TYPE "SSA_Germ_Par"	// UDT 2201
VERSION : 0.1
  STRUCT
   Switches1 : STRUCT
    StaOn24 : BOOL ;	//Example for comment: StaOn24WaterPumpA
    StaOn25 : BOOL ;
    StaOn26 : BOOL ;
    StaOn27 : BOOL ;
    StaOn28 : BOOL ;
    StaOn29 : BOOL ;
    StaOn30 : BOOL ;
    StaOn31 : BOOL ;
    StaOn16 : BOOL ;
    StaOn17 : BOOL ;
    StaOn18 : BOOL ;
    StaOn19 : BOOL ;
    StaOn20 : BOOL ;
    StaOn21 : BOOL ;
    StaOn22 : BOOL ;
    StaOn23 : BOOL ;
    StaOn08 : BOOL ;
    StaOn09 : BOOL ;
    StaOn10 : BOOL ;
    StaOn11 : BOOL ;
    StaOn12 : BOOL ;
    StaOn13 : BOOL ;
    StaOn14 : BOOL ;
    StaOn15 : BOOL ;
    StaOn00 : BOOL ;
    StaOn01 : BOOL ;
    StaOn02 : BOOL ;
    StaOn03 : BOOL ;
    StaOn04 : BOOL ;
    StaOn05 : BOOL ;
    StaOn06 : BOOL ;
    StaOn07 : BOOL ;
   END_STRUCT ;
   Switches2 : STRUCT
    StaOn24 : BOOL ;
    StaOn25 : BOOL ;
    StaOn26 : BOOL ;
    StaOn27 : BOOL ;
    StaOn28 : BOOL ;
    StaOn29 : BOOL ;
    StaOn30 : BOOL ;
    StaOn31 : BOOL ;
    StaOn16 : BOOL ;
    StaOn17 : BOOL ;
    StaOn18 : BOOL ;
    StaOn19 : BOOL ;
    StaOn20 : BOOL ;
    StaOn21 : BOOL ;
    StaOn22 : BOOL ;
    StaOn23 : BOOL ;
    StaOn08 : BOOL ;
    StaOn09 : BOOL ;
    StaOn10 : BOOL ;
    StaOn11 : BOOL ;
    StaOn12 : BOOL ;
    StaOn13 : BOOL ;
    StaOn14 : BOOL ;
    StaOn15 : BOOL ;
    StaOn00 : BOOL ;
    StaOn01 : BOOL ;
    StaOn02 : BOOL ;
    StaOn03 : BOOL ;
    StaOn04 : BOOL ;
    StaOn05 : BOOL ;
    StaOn06 : BOOL ;
    StaOn07 : BOOL ;
   END_STRUCT ;
   Values1 : STRUCT 	//Lineparameter data written by Host-System
    Value01 : DINT ;	//Example for comment: TurnoverTime [xxxs]
    Value02 : DINT ;
    Value03 : DINT ;
    Value04 : DINT ;
    Value05 : DINT ;
    Value06 : DINT ;
    Value07 : DINT ;
    Value08 : DINT ;
    Value09 : DINT ;
    Value10 : DINT ;
    Value11 : DINT ;
    Value12 : DINT ;
    Value13 : DINT ;
    Value14 : DINT ;
    Value15 : DINT ;
    Value16 : DINT ;
    Value17 : DINT ;
    Value18 : DINT ;
    Value19 : DINT ;
    Value20 : DINT ;
    Value21 : DINT ;
    Value22 : DINT ;
    Value23 : DINT ;
    Value24 : DINT ;
    Value25 : DINT ;
    Value26 : DINT ;
    Value27 : DINT ;
    Value28 : DINT ;
    Value29 : DINT ;
    Value30 : DINT ;
   END_STRUCT ;
   FlagSec : STRUCT
    Flag00 : BOOL ;
    Flag001 : BOOL ;
    Flag002 : BOOL ;
    Flag003 : BOOL ;
    Flag004 : BOOL ;
    Flag005 : BOOL ;
    Flag006 : BOOL ;
    Flag007 : BOOL ;
    Flag008 : BOOL ;
    Flag009 : BOOL ;
    Flag0010 : BOOL ;
    Flag0011 : BOOL ;
    Flag0012 : BOOL ;
    Flag0013 : BOOL ;
    Flag0014 : BOOL ;
    Flag0015 : BOOL ;
    Flag0016 : BOOL ;
    Flag0017 : BOOL ;
    Flag0018 : BOOL ;
    Flag0019 : BOOL ;
    Flag0020 : BOOL ;
    Flag0021 : BOOL ;
    Flag0022 : BOOL ;
    Flag0023 : BOOL ;
    Flag0024 : BOOL ;
    Flag0025 : BOOL ;
    Flag0026 : BOOL ;
    Flag0027 : BOOL ;
    Flag0028 : BOOL ;
    Flag0029 : BOOL ;
    Flag0030 : BOOL ;
    Flag0031 : BOOL ;
   END_STRUCT ;
   FlagGen : STRUCT
    WindAlarm : BOOL ;	//Wind speed is too high
    TurningStarted : BOOL ;	//Germination turning is started
    Underhorden_Clean_aktiv : BOOL ;	//Unterhordenreinigung aktiv
    WetStep : BOOL ;	//Active Step is Wet Step
    Flag004 : BOOL ;
    Flag005 : BOOL ;
    Flag006 : BOOL ;
    Flag007 : BOOL ;
    LOAD_VAL_HUB1 : BOOL ;	//Counter lifting device 1
    LOAD_VAL_HUB2 : BOOL ;	//Counter lifting device 2
    LOAD_VAL_DRIVE : BOOL ;	//Counter driving device
    LOAD_VAL_AFTER_FAILURE : BOOL ;	//Counter saved datas after failure
    Flag0012 : BOOL ;
    Flag0013 : BOOL ;
    Flag0014 : BOOL ;
    Flag0015 : BOOL ;
    InterlockedFunktionMode : BOOL ;
    ILO_CmdResetFault : BOOL ;
    Flag0018 : BOOL ;
    Flag0019 : BOOL ;
    Flag0020 : BOOL ;
    Flag0021 : BOOL ;
    Flag0022 : BOOL ;
    Flag0023 : BOOL ;
    Flag0024 : BOOL ;
    Flag0025 : BOOL ;
    Flag0026 : BOOL ;
    Flag0027 : BOOL ;
    Flag0028 : BOOL ;
    Flag0029 : BOOL ;
    Flag0030 : BOOL ;
    Flag0031 : BOOL ;
   END_STRUCT ;
   Spare140 : ARRAY  [148 .. 194 ] OF BYTE ;
   FlagMachine_0 : STRUCT 	//flags machine funktion
    FloorFwdPlus : BOOL ;	//Hordendrehrichtung Vorwärts, Rundenzaehler +1
    FloorFwdMinus : BOOL ;	//Hordendrehrichtung Vorwärts, Rundenzaehler -1
    FloorRevPlus : BOOL ;	//Hordendrehrichtung Rückwärts, Rundenzaehler +1
    FloorRevMinus : BOOL ;	//Hordendrehrichtung Rückwärts, Rundenzaehler -1
    OneShotGeenVrygVlr : BOOL ;	//Opkomende Flank geen vrijgave vloer
    HulpOneShotGeenVrygVlr : BOOL ;	//Hulp Opkomende Flank geen vrijgave vloer
    Flag006 : BOOL ;	//
    Flag007 : BOOL ;	//
    RotatPulseNotZero : BOOL ;	//
    ReducedSpeed : BOOL ;	//
    Speed2ndRound : BOOL ;	//Speed 2nd round during loading
    Flag013 : BOOL ;	//
    Flag014 : BOOL ;	//
    Flag015 : BOOL ;	//
    Flag016 : BOOL ;	//
    Flag017 : BOOL ;	//
    Flag020 : BOOL ;	//
    Flag021 : BOOL ;	//
    Flag022 : BOOL ;	//
    Flag023 : BOOL ;	//
    Flag024 : BOOL ;	//
    Flag025 : BOOL ;	//
    Flag026 : BOOL ;	//
    Flag027 : BOOL ;	//
    Flag030 : BOOL ;	//
    Flag031 : BOOL ;	//
    Flag032 : BOOL ;	//
    Flag033 : BOOL ;
    Flag034 : BOOL ;
    Flag035 : BOOL ;
    Flag036 : BOOL ;	//
    Flag037 : BOOL ;	//
   END_STRUCT ;
   ParIntProcess : STRUCT 	//Processparameter data
    UnloadungRounds : INT  := 2;
    LoadungRounds : INT  := 2;	//
    LoadingOverlap : INT  := 10;	//Impulse overlap by loading
    UnloadingOverlap : INT  := 20;	//Impulse overlap by unloading
    ReactTimeTempContr : S5TIME  := S5T#10S;	//Delay reaction temperature control below floor
    ReactTimeCO2Contr1 : S5TIME  := S5T#10S;	//Delay reaction CO2 control below floor
    BreakTimeFlapContr1 : S5TIME  := S5T#10S;	//Break time control fresh air flap
    DelayContrDelta_T : INT  := 10;	//Delay alarm control Delta-t in min
    DelayDeltaTemp : INT  := 2;	//Delay control Delta-t between temperature above and below floor, in min
    DelayMaxTemp : INT  := 2;	//Delay control temperature above below floor, in min
    Speed_ILO_FloorRotating : INT  := 22;	//Rotating speed floor from ILO-Rotating Floor Drives
    Speed_ILO_UnderCleaning : INT  := 80;	//Rotating speed floor from ILO-Floor Cleaning from below
    Speed_ILO_WallCleaning : INT  := 80;	//Rotating speed floor from ILO-WallCleaning
    ProcessActivVisuGerm : INT ;	//Display that Process is Active
    StateWordGerm : INT ;	//State-Number of the active Step
    TarPos_ILO_LiftDev : INT ;	//Target positon lifting devices from ILO-Mode
    TarPos_ILO_FreshAir : INT ;	//Target positon fresh air flap from ILO-Mode
    TarPos_ILO_RecycAir : INT ;	//Target positon recycling air flap from ILO-Mode
    Speed_ILO_Fan : INT ;	//Target speed germinatimng fan from ILO-Mode
    Speed_ILO_TravelDrive : INT ;	//Target speed travelling drive from ILO-Mode
    TarPos_ILO_WasteAir : INT ;	//Target positon waste air flap from ILO-Mode
    TargetTemperature_ILO : INT ;	//Target temperature from ILO-Mode
    Value23 : INT ;
    Value24 : INT ;
    Value25 : INT ;
    Value26 : INT ;
    Value27 : INT ;
    Value28 : INT ;
    Value29 : INT ;
    Value30 : INT ;
    Value31 : INT ;
    NextLevelLoading : INT ;	//Next level loading round
    Value33 : INT ;
    Value34 : INT ;
    Value35 : INT ;
    Value36 : INT ;
    CounterPosLoadingBeam : INT ;	//external counter beam position
    Value38 : INT ;
    Value39 : INT ;
    NumberOpenValves : INT ;	//number of opened spray valves air humidifikation
    SpeedProdSprayPump : INT ;	//setpoint speed pump product spray
    Value42 : INT ;
    Value43 : INT ;
    Value44 : INT ;
    PrevStep1stTurn : INT ;	//Store turning commands from prev. step
    PrevStep2ndTurn : INT ;	//Store turning commands from prev. step
    Value47 : INT ;
    Value48 : INT ;
    Value49 : INT ;
    ActualStep : INT ;	//Actual Step for visu
   END_STRUCT ;
   ParIntMachine : STRUCT 	//Machine parameter data
    ActualStep : INT ;	//Actual process step
    MAX_HUB_DIFF : INT  := 36;	//Max. Hubdifferenz zwischen Hubzug 1 + 2
    REINIGUNGSHOEHE : INT  := 100;	//Reinigungshoehe in mm
    MAX_SCHIEFLAGE : INT  := 150;	//Max. Schieflage zwischen Hubzug 1 + 2
    IMPULSE_HUBZUG1_OBEN : INT  := 480;	//Impulse : Hubantrieb 1 normieren bei Endpos.oben
    IMPULSE_HUBZUG2_OBEN : INT  := 480;	//Impulse : Hubantrieb 2 normieren bei Endpos.oben
    POSITION_HUBZUG1_OBEN : INT  := 1055;	//Hoehe in mm
    POSITION_HUBZUG2_OBEN : INT  := 1055;	//Hoehe in mm
    IMPULSE_RUNDE : INT  := 816;	//Impulse : Fahrantriebantrieb eine Runde (Diesen Wert bei der IBS ermitteln!!)
    SollwertFahrantrWenden : WORD  := W#16#DEF;	//21,7% von 100 Hz
    LiftDevMinPos : INT  := 100;	//Lifting device minimal position for rotation backwards
    FUELLHOEHE_PRODUKT : INT ;	//Produkt-Füllhöhe
    TargetPosTravDriveLoad : INT ;	//Soll-Position Fahrantrieb im Prozess
    RunTimeCleanDrive : S5TIME  := S5T#10M;	//Runing time drive floor cleaning from below
    DelayMonFlowContr : S5TIME  := S5T#10M;	//Delay monitoring flow control by loading
    RunTimeTurnScrews : INT  := 2;	//Time short run turning screws every 6 hours, in min
    LiftDevLowPos : INT  := 1000;	//Lifting device lowered position after turning round, in mm
    CutOffPointDosing : INT ;	//Cut-off point dosing
    GerminatingBoxNumber : INT ;
    TargetPosTravDriTurnLeft : INT ;
    TargetPosTravDriTurnRigt : INT ;
    TargetPosTravDriveUnload : INT ;
    Help1StartTurning : INT ;	//hulpwoord 1 tbv  wenderen
    Resetbreaktime : INT ;	//tbv resetten wenderpauze
    Help2StartTurning : INT ;	//hulpwoord 2 tbv  wenderen
    TurningHourOneOrTwo : INT ;	//wenderuur 1 of 2
    Timer_tbv_opk_wend_spr : INT ;	//timer tbv het opkomen van het wenderen of sproeien
    TargetPosFreshAir : INT ;	//Target position fresh air flap/jalousie/louver
    TargetPosRecyclingAir : INT ;	//Target position recycling air flap/jalousie/louver
    TargetPosWasteAir : INT ;	//Target position waste air flap/jalousie/louver
    TargetSpeedGermFan : INT ;	//Target speed fan germinating box
    TargetSpeedLoadScrew : INT ;	//Target speed loading/unloading screw germinating box
    Value33 : INT ;
    Value34 : INT ;
    Value35 : INT ;
    Value36 : INT ;
    Value37 : INT ;
    HulpwoordTbvTelpulsbewak : INT ;	//Hulpwoord tbv telpulsbewaking vloer
    PresetWaardeTimerTelpVlR : INT ;	//Preset waarde van timer tbv telpulsbewaking vloer.
    GemiddeldeHoogteHefwerk : INT ;	//De gemiddelde hoogte van de hefwerken
    GewensteOntlaadhoogte : INT ;	//Gewenste Ontlaadhoogte Hefwerken
    Value42 : INT ;
    Value43 : INT ;
    Value44 : INT ;
    Value45 : INT ;
    Value46 : INT ;
    Value47 : INT ;
    Value48 : INT ;
    GrowingOffset : INT ;
    LastLoadingLevel : INT ;
   END_STRUCT ;
   FlagFunction_0 : STRUCT 	//Flags section
    FlagLoadingFinishedFP : BOOL ;	//
    FlagFirstTurning : BOOL ;	//First turning round after loading
    FlagNextStep : BOOL ;
    FlagLoadingFinished : BOOL ;
    StartTurningForMGR : BOOL ;	//Enable start turning for group control
    Inf29 : BOOL ;
    FlagLoadingOverlap : BOOL ;
    FlagUnloadingOverlap : BOOL ;
    ImpulsUnloadLevelReached : BOOL ;	//Unloading level has been reached
    UnloadLevelReachedFP : BOOL ;	//FP unloading level has been reached
    ShortRunTurnScrews : BOOL ;	//Short run turning screws every 6 hours
    LowerLiftDevAfterTurn : BOOL ;	//To lower lifting device after every turning round
    UnloadingLevelAdjusted : BOOL ;	//
    FlagWallCleanStopFP : BOOL ;	//
    Spare2 : BOOL ;	//
    FlagLoadingStartedFP : BOOL ;
    ImpulseLoadingStarted : BOOL ;
    FlagUnloadingStartedFP : BOOL ;
    ImpulseUnloadingStarted : BOOL ;
    FlagCleaningStartedFP : BOOL ;
    ImpulseCleaningStarted : BOOL ;
    FlagTurningStartedFP : BOOL ;
    ImpulseTurningStarted : BOOL ;
    FlagTurningStartedRight : BOOL ;
    FlagTurningStartedLeft : BOOL ;
    FlagStep14FN : BOOL ;
    ImpulseUnloadFirstPart : BOOL ;
    FlagStepFirstTurning : BOOL ;	//First turning round in this step is finished
    FlagStepSecondTurning : BOOL ;	//Second turning round in this step is finished
    ReleaseUnloadFirstPart : BOOL ;
    InfReleaseUnloading : BOOL ;
   END_STRUCT ;
   FlagMachine : STRUCT 	//flags machine funktion
    Hubzug1_Low : BOOL ;	//Hubzug 1 Richtungsvorwahl senken
    Hubzug1_High : BOOL ;	//Hubzug 1 Richtungsvorwahl heben
    Hubzug2_Low : BOOL ;	//Hubzug 2 Richtungsvorwahl senken
    Hubzug2_High : BOOL ;	//Hubzug 2 Richtungsvorwahl heben
    Stop_Hubzuege : BOOL ;	//Differenz Hub1-Hub2>Vorgabewert
    Hubzug1_Speed_Ctr : BOOL ;	//Hubantrieb 1 innen Drehueberwachung
    Hubzug2_Speed_Ctr : BOOL ;	//Hubantrieb 2 aussen Drehueberwachung
    Hubzuege_ueber_MinPos : BOOL ;	//Hubzug 1 und Hubzug 2 mehr als 100mm ueber ihrer Nullposition
    Hubzug1_Stop_NullPos_man : BOOL ;	//Hoehe Hubzug 1 <= NULL-Position
    Hubzug2_Stop_NullPos_man : BOOL ;	//Hoehe Hubzug 2 <= NULL-Position
    Hubdiff1_2 : BOOL ;	//Hubdifferenz Hub1 > Hub2
    Hubdiff2_1 : BOOL ;	//Hubdifferenz Hub2 > Hub1
    Hubzug1_Hoch : BOOL ;	//Hubzug 1 Isthoehe > 300mm (Freigabe Ausraeumglocke schliessen) und Hubzuege heb
    Hubzug2_Hoch : BOOL ;	//Hubzug 2 Isthoehe > 300mm (Freigabe Ausraeumglocke schliessen) und Hubzuege heb
    Start_Hubzuege_Heben : BOOL ;	//Hubzuege heben
    Hubdiff1_2_NegAlt : BOOL ;	//Hubdifferenz Hub1 > Hub2 Alt-Signal
    Hubdiff1_2_NegFlag : BOOL ;	//Hubdifferenz Hub1 > Hub2 Flanken-Signal
    Hubdiff2_1_NegAlt : BOOL ;	//Hubdifferenz Hub2 > Hub1 Alt-Signal
    Hubdiff2_1_NegFlag : BOOL ;	//Hubdifferenz Hub2 > Hub1 Flanken-Signal
    Fahrantrieb_Speed_Ctr1 : BOOL ;	//Fahrantrieb Drehueberwachung
    Fahrantrieb_Start_ok : BOOL ;	//Es sind weniger als 2 Fahrantriebe nicht gestartet
    Fahrantrieb_FU_Fault : BOOL ;	//Sammelstörung von allen 12 FU's
    Fahrantriebe_Fwd_Rev : BOOL ;	//Aktuelle Drehrichtung Fahrantriebe (0=Fwd; 1=Rev)
    Fahrantriebe_Vorwaerts : BOOL ;	//Fahrantriebe Ausgang Richtung Vorwärts
    Fahrantriebe_Rueckwaerts : BOOL ;	//Fahrantriebe Ausgang Richtung Rückwärts
    NULL_INDEX_FP : BOOL ;
    ImpulsNullstellung : BOOL ;
    ImpulsNullstellungFP : BOOL ;
    WEGMESSUNG_0 : BOOL ;
    WEGMESSUNG_0_FLAG : BOOL ;
    HubzuegeUeberProdukt : BOOL ;	//Schnecke ueber Produktschicht
    HubzuegeParkposition : BOOL ;	//Beide Hubzuege in Parkposition
   END_STRUCT ;
   FlagFunction_1 : STRUCT 	//Flags functions
    StepLoading : BOOL ;	//Function Loading is active
    StepUnloading : BOOL ;	//Function Unloading is active
    StepCleaning : BOOL ;	//Function Cleaning is active
    LoadingBreak : BOOL ;	//Function Loading is interrupted
    UnloadingBreak : BOOL ;	//Function Unloading is interrupted
    CleaningBreak : BOOL ;	//Function Cleaning is interrupted
    FinishLoading : BOOL ;	//Function Loading is finished
    FinishUnloading : BOOL ;	//Function Unloading is finished
    FinishCleaning : BOOL ;	//Function Cleaning is finished
    LoadingStarted : BOOL ;	//Germination loading is started
    UnloadingStarted : BOOL ;	//Germination unloading is started
    CleaningStarted : BOOL ;	//Germination cleaning is started
    Round_1 : BOOL ;	//Fahrantrieb 1.Runde
    Round_2 : BOOL ;	//Fahrantrieb 2.Runde
    Round_3 : BOOL ;	//Fahrantrieb 3.Runde
    Round_4 : BOOL ;	//Fahrantrieb 4.Runde
    Round_5 : BOOL ;	//Fahrantrieb 5.Runde
    Round_6 : BOOL ;	//Fahrantrieb 6.Runde
    Beladung_beendet : BOOL ;	//Fahrantrieb; Beladung_beendet
    Entladerunden_erreicht : BOOL ;	//Fahrantrieb; Entladerunden erreicht
    Reinigungsrunde_erreicht : BOOL ;	//Fahrantrieb; Reinigungsrunde erreicht
    TurningStart : BOOL ;	//Start turning
    TurningStop : BOOL ;	//Stop turning
    TurningLeft : BOOL ;	//Germination turning left
    TurningRight : BOOL ;	//Germination turning right
    LoadFirstPartEnd : BOOL ;	//Grundschicht ist bedeckt, prozess kann starten
    TurningWithSpraying : BOOL ;	//Turning-round in this step with spraying
    TurningWithoutSpraying : BOOL ;	//Turning-round in this step without spraying
    UnloadFirstPartEnd : BOOL ;	//First half of germinating box is unloaded
    UnloadSecondPartEnd : BOOL ;	//Second half of germinating box is unloaded
    UnloadFirstPart : BOOL ;	//Unload first half of germinating box
    UnloadSecondPart : BOOL ;	//Unload second half of germinating box
   END_STRUCT ;
   FlagProcess : STRUCT 	//Flags process
    ProcessActive : BOOL ;	//Process is active
    ProcessStartFP : BOOL ;	//Flank start process
    ProcessStartScan : BOOL ;	//Impulse first step
    MessageNoNextStep : BOOL ;	//Message "No next step"
    FP_SendResultToPIC : BOOL ;
    Vraag_menu_wenderen : BOOL ;	//Vraag vanuit het recept om te wenderen
    Vraag_menu_sproeien : BOOL ;	//Vraag vanuit het recept om te sproeien
    Vraag_menu_doseren : BOOL ;	//Vraag vanuit het recept om te doseren
    FlagWallCleanStartFP : BOOL ;	//Hulp one shot wandreinigen gestart
    ImpulseWallCleanStarted : BOOL ;	//One shot wandreinigen gestart
    Inf18 : BOOL ;
    VrijgaveWenderFunctie : BOOL ;	//Geen vrijgave om wenderbits in FC2019 aan te zetten
    Aussenluft_zu_warm : BOOL ;
    Cooling : BOOL ;
    AirHumidificationValve1 : BOOL ;
    AirHumidificationValve2 : BOOL ;
    Breakpoint_Aktiv : BOOL ;
    ProcessEnd : BOOL ;
    Cooling_Activ : BOOL ;
    Abkuehlen : BOOL ;
    Inf24 : BOOL ;
    Vent_ReglerAusg_Plus : BOOL ;
    Vent_ReglerAusg_PlusFP : BOOL ;
    Vent_ReglerAusg_Minus : BOOL ;
    Vent_ReglerAusg_MinusFP : BOOL ;
    Ventilator_Drehzahl_HH : BOOL ;	// Drehzahlbereich HH [85 - 100%]
    Ventilator_Drehzahl_H : BOOL ;	// Drehzahlbereich  H [65 -  84%]
    Ventilator_Drehzahl_L : BOOL ;	// Drehzahlbereich  L [55 -  64%]
    Ventilator_Drehzahl_LL : BOOL ;	// Drehzahlbereich LL [40 -  54%]
    VentilatorDrehzahlMin : BOOL ;
    VentilatorDrehzahlMax : BOOL ;
    Inf37 : BOOL ;
   END_STRUCT ;
   FlagProcess1 : STRUCT 	//Flags process
    FreshAirFlapCLOSE : BOOL ;	//Close fresh air flap
    FreshAirFlapOPEN : BOOL ;	//Open fresh air flap
    ControlFreshAirFlap : BOOL ;	//Control fresh air flap
    ControlFlap_OPEN : BOOL ;	//Control - fresh air flap 1% open
    ControlFlap_CLOSE : BOOL ;	//Control - fresh air flap 1% close
    ControlTemperature : BOOL ;	//Priority temperature for control fresh air flap
    ControlCO2 : BOOL ;	//Priority CO2 for control fresh air flap
    BasicPosFreshAirFlap : BOOL ;	//Fresh air flap in basic position
    ExhaustAirFlap_1_CLOSE : BOOL ;	//Close exhaust air flap 1
    ExhaustAirFlap_1_OPEN : BOOL ;	//Open exhaust air flap 1
    BasicPosExhaustAirFlap_1 : BOOL ;	//Exhaust air flap 1 in basic position
    ExhaustAirFlap_2_CLOSE : BOOL ;	//Close exhaust air flap 2
    ExhaustAirFlap_2_OPEN : BOOL ;	//Open exhaust air flap 2
    BasicPosExhaustAirFlap_2 : BOOL ;	//Exhaust air flap 2 in basic position
    DeltaTempPlus : BOOL ;	//
    DeltaTempMinus : BOOL ;	//
    InterlockedFunktionMode : BOOL ;	//
    Inf21 : BOOL ;	//
    Inf22 : BOOL ;	//
    Inf23 : BOOL ;	//
    Inf24 : BOOL ;	//
    Inf25 : BOOL ;	//
    DeltaTempNextStep : BOOL ;	//Delta Temperature go to next step
    MaxTempNextStep : BOOL ;	//Max Temperature above floor go to next step
    FlankeStartRecept_IN : BOOL ;	//ONE_SHOT_START_RECEPT
    PT100Defect_IN : BOOL ;	//PT100_boven_vloer_stuk
    FreigabeStartRezept_IN : BOOL ;	//VRIJGAVE_START_RECEPT
    tm_Frequenzregler_IN : BOOL ;	//wanneer ventilator in bedrijf meldt
    Flanke_FreigabeRezept_IO : BOOL ;	//One_shot_vent_op_basis
    HandAutoVentilator_IO : BOOL ;	//Hand_automaat_kiemvent
    Inf36 : BOOL ;	//
    TurnWithClean : BOOL ;	//Turning with floor cleaning from below
   END_STRUCT ;
   FlagProcess2 : STRUCT 	//Flags process
    Turning1WithSpraying : BOOL ;	//First turning round in this step with spraying
    Turning1WithDosing : BOOL ;	//First turning round in this step with spraying and dosing
    Turning1WithoutSpraying : BOOL ;	//First turning round in this step without spraying
    Turning2WithSpraying : BOOL ;	//Second turning round in this step with spraying
    Turning2WithDosing : BOOL ;	//Second turning round in this step with spraying and dosing
    Turning2WithoutSpraying : BOOL ;	//Second turning round in this step without spraying
    MinBreakTimeFinish : BOOL ;	//Minimal break time is finished
    MaxBreakTimeFinish : BOOL ;	//Maximal break time is finished
    ReleaseSpraying : BOOL ;	//Release spraying for this germinating box
    ReleaseDosing : BOOL ;	//Release dosing for this germinating box
    Delta_T : BOOL ;	//Delta-t is > or < recipe value
    StartSpraying : BOOL ;	//Store impulse start spraying
    HighWindForce : BOOL ;	//Wind force too high
    ReleaseTurning : BOOL ;	//Release turning for this germinating box
    StartFirstTurningRound : BOOL ;	//Store impulse for start first turning round acc. recipe
    StartSecondTurningRound : BOOL ;	//Store impulse for start second turning round acc. recipe
    PauseBeforeSpraying_FP : BOOL ;	//
    PauseBeforeSpraying_IMP : BOOL ;
    PauseBeforeSprayingFin : BOOL ;	//Pause before spraying is finished
    AlarmControlDelta_T : BOOL ;	//Alarm control Delta-t
    StartFirstTurningFP : BOOL ;
    StartSecondTurningFP : BOOL ;	//
    StartFirstSprayingFP : BOOL ;
    StartFirstDosingFP : BOOL ;
    StartSecondSprayingFP : BOOL ;
    StartSecondDosingFP : BOOL ;
    StartFirstSpraying : BOOL ;	//Store impulse for start first turning round with spraying acc. recipe
    StartFirstDosing : BOOL ;	//Store impulse for start first turning round with dosing acc. recipe
    StartSecondSpraying : BOOL ;	//Store impulse for start second turning round with spraying acc. recipe
    StartSecondDosing : BOOL ;	//Store impulse for start second turning round with dosing acc. recipe
    Sonderwenden : BOOL ;	//Sonderwenden
    FaultDB_Copy : BOOL ;	//Fault DB Copy FC49
   END_STRUCT ;
   ProcessValue : STRUCT 	//Process values, used only in the PLC
    Value01 : DINT ;
    Value02 : DINT ;
    Value03 : DINT ;
    SetpointDeltaTempDint : DINT ;
    ActValueDeltaTempDint : DINT ;
    ActValMaxTempAboveDint : DINT ;
    ResultDeltaTemp : DINT ;
    ConsumptionWater : DINT ;	//Water consumption per section
    CurrentConsumCoolEnergy : DINT ;	//Aktueller Verbrauch Kühl-Energie
    ConsumptionCoolingEnergy : DINT ;	//Verbrauchte Menge Kühl-Energie
    LevelGlycol : DINT ;	//something with glycol
    Profimess_Command : DINT ;	//command to read data from Profimess
    Value13 : DINT ;
    Value14 : DINT ;
    Value15 : DINT ;
    Value16 : DINT ;
    HelpConsumptionwater : DINT ;	//Tussenwoord voor opslag aantal M3 sproeien
    RET_VAL_BreakTime : INT ;
    StepNrActCopy : INT ;
    StartStepAct : DATE_AND_TIME ;
    ActualTime : DATE_AND_TIME ;
    BreakTime : DATE_AND_TIME ;
    StartCooling : DATE_AND_TIME ;
    StepTimeAct : TIME ;
    BreakTimeAct : TIME ;
    TimeControlDelta_T : TIME ;
    PauseBeforeSpraying : TIME ;
   END_STRUCT ;
   ProcessValueReal : STRUCT 	//Process real values, used only in the PLC
    SpeedVentilatorBasic : REAL ;	//Setpoint Fanspeed in %
    PositFreshAirFlapBasic : REAL ;	//Setpoint basic flap position
    ActTempBelowFloor : REAL ;	//Actual temperature below floor
    TargTempBelowFloor : REAL ;	//Setpoint temperature below floor
    ActTempAboveFloor : REAL ;	//Actual temperature above floor
    TargTempAboveFloor : REAL ;	//Setpoint temperature above floor
    NivoDoseertank : REAL ;	//Nivo doseertank in real
    Value08 : REAL ;	//
    Value09 : REAL ;	//
    Value10 : REAL ;	//
    Value11 : REAL ;	//
    Value12 : REAL ;	//
    Value13 : REAL ;	//
    Value14 : REAL ;
    Value15 : REAL ;
    Value16 : REAL ;
    Value17 : REAL ;
    Value18 : REAL ;
    Value19 : REAL ;
    Value20 : REAL ;
    CoolingEnergyAct : REAL ;
    CoolingEnergySum : REAL ;
    Value23 : REAL ;
    Value24 : REAL ;
    Profimess_Wirkleistung : REAL ;
    Profimess_Blindleistung : REAL ;
    Profimess_Frequenz : REAL ;
    Profimess_Wirkleist_Psec : REAL ;
    Profimess_Arbeit_Batch : REAL ;
    EnergieKWs : REAL ;
   END_STRUCT ;
   MachineValue : STRUCT 	//Machine values, used only in the PLC
    ISTWERT_FAHRANTRIEB_POSI : INT ;	//Ist-Position Fahrantrieb
    FAHRANTRIEB_UMDREHUNGEN : INT ;	//Rundenzaehler Fahrantrieb
    IST_HUB_DIFF : INT ;	//Istwert Hubdifferenz zwischen Hubzug 1 + 2
    ISTWERT_HUBZUG1_Z_IMP : INT ;	//Istwert Zaehlimpulse Hubzug 1
    ISTWERT_HUBZUG2_Z_IMP : INT ;	//Istwert Zaehlimpulse Hubzug 2
    SCHRAEGE_HUB1_HUB2 : INT ;	//Schraege Hub 1 > Hub 2
    SOLLWERT_HUBZUG1_HOEHE : INT ;
    SOLLWERT_HUBZUG2_HOEHE : INT ;
    ISTWERT_HUBZUG1_HOEHE : INT ;
    ISTWERT_HUBZUG2_HOEHE : INT ;
    SCHRAEGE_HUB1_MINUS_HUB2 : INT ;	//Schraege Hub 1 minus Hub 2
    SCHRAEGE_HUB2_MINUS_HUB1 : INT ;	//Schraege Hub 2 minus Hub 1
    BELADERUNDEN_START_HUB : INT ;	//Anhebeposition in Grad
    ISTWERT_FAHRANTRIE_Z_IMP : INT ;	//Istwert Zaehlimpulse Fahrantrieb
    Fahrantriebe_Gestartet : INT ;	//Zaehlwert der gestarteten Fahrantriebe
    SollwertFahrantrieb : WORD ;	//an FU
    Fahrzeit_Reinigungswagen : INT ;	//Fahrzeit des Reinigungswagens unter der Horde
    Position_Reinigungswagen : INT ;	//Position der Reinigungswagens unter der Horde
    ISTWERT_HUBZUG1_DOPPEL : DINT ;	//Hubzug 1 : Hoehe [mm] Rechenwert
    ISTWERT_HUBZUG2_DOPPEL : DINT ;	//Hubzug 2 : Hoehe [mm] Rechenwert
    BELADERUNDEN_HUB_IMP : DINT ;	//Anhebeposition in Pulsen
    FAHR_GRAD_DOPPEL : DINT ;	//Fahrantrieb : Umdrehung in Grad Rechenwert
    RotatingSpeed : DINT ;	//Rotating Speed temp
    FloorPosAbs : DINT ;	//Floor absolute position
    FloorPositionPercent : DINT ;	//Floor position percentagewise
    RotatingPulseAbsolut : DINT ;
    RondgangWenderenSproeien : DINT ;	//Floor position percentagewise tbv nieuwe functie wenderen sproeien H.v.L.
    MinimaleOntlaadSnelheid : DINT ;	//De minimale ontlaadsnelheid van de vloer
    HulpwoordtTelStandVloer : DINT ;	//HulpwoordTellerstand Vloer
    Value21 : DINT ;
    Value22 : DINT ;
    Value23 : DINT ;
    Value24 : DINT ;
    Value25 : DINT ;
    Value26 : DINT ;
    Value27 : DINT ;
    HUBZUG1_Z_IMP_HOLD : DINT ;	//Istwert Zaehlimpulse Hubzug 1 gespeichert
    HUBZUG2_Z_IMP_HOLD : DINT ;	//Istwert Zaehlimpulse Hubzug 2 gespeichert
    FAHRANTRIEB_Z_IMP_HOLD : DINT ;	//Istwert Zaehlimpulse Fahrantrieb gespeichert
   END_STRUCT ;
   MachineValueReal : STRUCT 	//Machine real values, used only in the PLC
    HUB1_MM_PRO_IMPULS : REAL  := 2.197917e+000;	//Hubzug 1 : Hoehe [mm] pro Hubimpuls
    HUB2_MM_PRO_IMPULS : REAL  := 2.197917e+000;	//Hubzug 2 : Hoehe [mm] pro Hubimpuls
    FAHRANTRIEB_IMP_GRAD : REAL  := 4.411765e-001;	//Winkelgrad pro Fahrimpuls (wird automatisch berechnet)
    FAHR_GRAD_PRO_IMPULS : REAL ;	//Fahrantrieb : Umdrehung in Grad pro Fahrimpuls Real-Rechenwert
    IMPULSE_RUNDE_REAL : REAL ;	//Impulse : Fahrantrieb eine Runde Real-Rechenwert
    Faktor_Reinigungswagen_R : REAL ;	//Weg/Zeit-Faktor Reinigungswagens unter der Horde
    Fahrzeit_Reinigungswag_R : REAL ;	//Fahrzeit der Reinigungswagens unter der Horde
    Position_Reinigungswag_R : REAL ;	//Position der Reinigungswagens unter der Horde
    FAHRANTRIEB_IMP_PROZ : REAL ;	//Prozentzahl pro Fahrimpuls (wird automatisch berechnet)
    BELADERUNDEN_START_HUB : REAL ;	//Anhebeposition von % in Grad
    Value11 : REAL ;
    Value12 : REAL ;
    Value13 : REAL ;
    Value14 : REAL ;
    Value15 : REAL ;
    Value16 : REAL ;
    Value17 : REAL ;
    Value18 : REAL ;
    Value19 : REAL ;
    Value20 : REAL ;
    Value21 : REAL ;
    Value22 : REAL ;
    Value23 : REAL ;
    Value24 : REAL ;
    Value25 : REAL ;
    Value26 : REAL ;
    Value27 : REAL ;
    Value28 : REAL ;
    Value29 : REAL ;
    Value30 : REAL ;
   END_STRUCT ;
   Spare892 : INT ;
   Spare894 : INT ;
   Error : STRUCT
    Value : INT ;
    Bit : BOOL ;
   END_STRUCT ;
  END_STRUCT ;	
END_TYPE

TYPE "SSA_Germ_Recipe"	// UDT 2202
VERSION : 0.1
  STRUCT
   RecipeHeader : UDT 2204;
   Step : ARRAY  [1 .. 28 ] OF UDT 2205;
  END_STRUCT ;	
END_TYPE

TYPE "SSA_Germ_Analog"	// UDT 2203
VERSION : 0.1
  STRUCT
   SpeedVentilatorBasic : INT ;	//Setpoint Fanspeed in %
   PositFreshAirFlapBasic : INT ;	//Setpoint basic flap position
   spare04 : INT ;
   spare06 : INT ;
   spare08 : INT ;
   spare10 : INT ;
   spare12 : INT ;
   spare14 : INT ;
   spare16 : INT ;
   spare18 : INT ;
   spare20 : INT ;
   spare22 : INT ;
   spare24 : INT ;
   spare26 : INT ;
   spare28 : INT ;
   spare30 : INT ;
   spare32 : INT ;
   spare34 : INT ;
   Change : STRUCT
    SpeedVentilatorBasicGer : BOOL ;	//the analog value has change if there is a bit
    PositFreshAirFlapBasic : BOOL ;	//the analog value has change if there is a bit
    NumberOfAeriationLines : BOOL ;	//the analog value has change if there is a bit
    DelayNextValve : BOOL ;	//the analog value has change if there is a bit
    DelayNextAeriationCycle : BOOL ;	//the analog value has change if there is a bit
    SpeedVentilator1 : BOOL ;	//the analog value has change if there is a bit
    SpeedVentilator2 : BOOL ;	//the analog value has change if there is a bit
    SpeedVentilator3 : BOOL ;	//the analog value has change if there is a bit
    SpeedVentilator4 : BOOL ;	//the analog value has change if there is a bit
    DrainTimeWaterAeriation : BOOL ;	//the analog value has change if there is a bit
    DrainTimeWaterCO2Suck : BOOL ;	//the analog value has change if there is a bit
    StartSpraying : BOOL ;	//the analog value has change if there is a bit
    TimeSpraying : BOOL ;	//the analog value has change if there is a bit
    DelaySpraying : BOOL ;	//the analog value has change if there is a bit
    SpeedVentilatorBasicKiln : BOOL ;	//the analog value has change if there is a bit
    PositWasteAirFlapBasic : BOOL ;	//the analog value has change if there is a bit
    PositRecyclAirIFlapBasic : BOOL ;	//the analog value has change if there is a bit
    PositRecyclAirDFlapBasic : BOOL ;	//the analog value has change if there is a bit
    SpeedRotatingFloorDrives : BOOL ;	//the analog value has change if there is a bit
    spare_20 : BOOL ;
    spare_21 : BOOL ;
    spare_22 : BOOL ;
    spare_23 : BOOL ;
    spare_24 : BOOL ;
    spare_25 : BOOL ;
    spare_26 : BOOL ;
    spare_27 : BOOL ;
    spare_28 : BOOL ;
    spare_29 : BOOL ;
    spare_30 : BOOL ;
    spare_31 : BOOL ;
    spare_32 : BOOL ;
   END_STRUCT ;
  END_STRUCT ;	
END_TYPE

TYPE "SSA_Germ_Recipe_Header"	// UDT 2204
VERSION : 0.1
  STRUCT
   NumberOfSteps : INT  := 20;	//Number of steps
   Duration_Germinating : DINT ;	//Estimated duration Germinating
   OutsideTempSwitchpoint_1 : DINT ;	//Switchpoint 1 Outside Temperature additional fresh air
   OutsideTempSwitchpoint_2 : DINT ;	//Switchpoint 2 Outside Temperature additional fresh air
   AdditonalTurnByTempDev : DINT ;	//Additional turning round due to teperature deviation above floor in °C
   AlarmOverTempAboveFloor : DINT ;	//Switchpoint Alarm Over-Temperature above floor in °C
   AlarmUnderTempAboveFloor : DINT ;	//Switchpoint Alarm Under-Temperature above floor in °C
   SPARE_DINT003 : DINT ;
   MinimalDelayNextTurn : INT ;	//Minimal time between two starts of turning rounds in min
   StepCleanBelowFloor : INT ;	//Stepnumber to clean floorconstruction from below during first turning round
   DelayNextTurning : INT ;	//Delay to next turning-round in actual step
   FreshAirValueLimit_1 : INT ;	//Limit 1 open fresh air outlet in %
   FreshAirValueLimit_2 : INT ;	//Limit 2 open fresh air outlet in %
   Loading : UDT 2011;
   Unloading : UDT 2012;
   Cleaning : UDT 2013;
  END_STRUCT ;	
END_TYPE

TYPE "SSA_Germ_Step"	// UDT 2205
VERSION : 0.1
  STRUCT
   StepNumber : INT  := 1;
   StepType : INT  := 1;	//Type Loading = 0;Germinating = 1;Unloading = 4;Cleaning = 8
   NextStep : INT  := 2;	//Nr.1 to 28=processsteps;Nr.101= unloading 1.part;Nr.102= unloading 2.part;
   StepTime_Min : INT ;	//Minimal Steptime in h
   StepTime_Max : INT ;	//Maximal Steptime in h
   TemperaturBelowFloor : DINT ;	//Setpoint Temperature in °C
   TemperaturAboveFloor : DINT ;	//Setpoint Temperature in °C
   WarningTempAboveFloor : DINT ;	//Setpoint Temperature in °C
   DeltaTempSwitchpointAir : DINT ;	//Switchpoint Delta Temperature additional fresh air in °C
   CO2SwitchpointAir : DINT ;	//Switchpoint CO2 additional fresh air in °C
   Moisture : DINT ;	//Setpoint air-moisture below floor (not used)
   DeltaTempSwitchpointStep : DINT ;	//Switchpoint Delta Temperature go to next step in °C
   MaxTempAboveFloorStep : DINT ;	//Switchpoint Temperature above floor go to next step in °C
   VolumeSprayingWaterR_1 : DINT ;	//Volume of spraying water in one turning round in m³
   VolumeSprayingAcidR_1 : DINT ;	//Volume of acid in one turning round with spraying and dosing in l
   WarningMaxTempAboveFloor : DINT ;	//Setpoint Temperature in °C Delta Temp
   WarningMinTempBelowFloor : DINT ;	//Setpoint Temperature in °C Delta Temp
   VolumeSprayingWaterR_2 : DINT ;	//Volume of spraying water in one turning round in m³
   VolumeSprayingAcidR_2 : DINT ;	//Volume of acid in one turning round with spraying and dosing in l
   SpeedVentilatorBasic : INT ;	//Setpoint Fanspeed in %
   SpeedVentilatorMaximal : INT ;	//Setpoint Fanspeed in % (not used)
   PosFreshAirFlapBasic : INT ;	//Setpoint basic flap position in %
   PosFreshAirFlapMax : INT ;	//Setpoint maximal flap position in % (GMC)
   PosWasteAirFlapBasic : INT ;	//Setpoint basic flap position in % (GMC)
   spare76 : INT ;
   StartTurningRound_1 : INT ;	//Starttime first turning-round in this step im h
   StartTurningRound_2 : INT ;	//Starttime second turning-round in this step im h
   spare82 : INT ;
   MaxDelayNextTurning : INT ;	//Maximum delay to next Turning-round in h
   SPARE_INT001 : INT ;
   SPARE_INT002 : INT ;
   SPARE_INT003 : INT ;
   Cooling : BYTE ;	//Activate Cooling System y/n (1/0)
   AirMoisten : BYTE ;	//Moisten Air y/n (1/0)
   SPARE_BYTE000 : BYTE ;	//
   TurningWithSpraying_1 : BYTE ;	//First turning-round in this step with spraying y/n (1/0)
   TurningWithDosing_1 : BYTE ;	//First turning-round in this step with spraying and dosing y/n (1/0)
   TurningWithSpraying_2 : BYTE ;	//Second turning-round in this step with spraying y/n (1/0)
   TurningWithDosing_2 : BYTE ;	//Second turning-round in this step with spraying and dosing y/n (1/0)
   SPARE_BYTE001 : BYTE ;
  END_STRUCT ;	
END_TYPE

TYPE "SSA_Kiln_Cmd"	// UDT 2300
VERSION : 0.1
  STRUCT
   Functions : STRUCT
    StartLoading : BOOL ;	//Start Function Loading
    BreakLoading : BOOL ;	//Break Function Loading
    ContinueLoading : BOOL ;	//Continue Function Loading
    StopLoading : BOOL ;	//Stop Function Loading
    UnloadingManuel : BOOL ;	//Unloading in Manuel Mode, only for Kiln
    StartUnloading : BOOL ;	//Start Function Unloading
    BreakUnloading : BOOL ;	//Break Function Unloading
    ContinueUnloading : BOOL ;	//Continue Function Unloading
    StopUnloading : BOOL ;	//Stop Function Unloading
    StartCleaning : BOOL ;	//Start Function Cleaning
    BreakCleaning : BOOL ;	//Break Function Cleaning
    ContinueCleaning : BOOL ;	//Continue Function Cleaning
    CleaningReady : BOOL ;	//Stop Function Cleaning
    StartProcess : BOOL ;	//Comand of Future
    Comand16 : BOOL ;
    Comand17 : BOOL ;
   END_STRUCT ;
   General : STRUCT
    LiftingDeviceUP : BOOL ;	//Lifting device UP
    LiftingDeviceDOWN : BOOL ;	//Lifting device DOWN
    LiftingDeviceSTOP : BOOL ;	//Lifting device STOP
    LiftingDeviceRESET : BOOL ;	//Lifting device RESET FAULT
    LoadUnloadScrewINSIDE : BOOL ;	//Loading-Unloading Screw INSIDE (LEFT)
    LoadUnloadScrewOUTSIDE : BOOL ;	//Loading-Unloading Screw OUTSIDE (RIGHT)
    LoadUnloadScrewSTOP : BOOL ;	//Loading-UnloadingScrew STOP
    LoadUnloadScrewRESET : BOOL ;	//Loading-UnloadingScrew RESET FAULT
    DischargeFlapOPEN : BOOL ;	//Discharge flap OPEN
    DischargeFlapCLOSE : BOOL ;	//Discharge flap CLOSE
    DischargeFlapRESET : BOOL ;	//Discharge flap RESET FAULT
    RotatingFloorDrivesRIGHT : BOOL ;	//Rotating Floor Drives RIGHT
    RotatingFloorDrivesLEFT : BOOL ;	//Rotating Floor Drives LEFT
    RotatingFloorDrivesSTOP : BOOL ;	//Rotating Floor Drives STOP
    RotatingFloorDrivesRESET : BOOL ;	//Rotating Floor Drives RESET FAULT
    spare_16 : BOOL ;
   END_STRUCT ;
   SPARE0 : BYTE ;
   SPARE1 : BYTE ;
   SPARE2 : BYTE ;
   SPARE3 : BYTE ;
   SPARE4 : BYTE ;
   SPARE5 : BYTE ;
  END_STRUCT ;	
END_TYPE

TYPE "SSA_Kiln_Par"	// UDT 2301
VERSION : 0.1
  STRUCT
   Switches1 : STRUCT
    StaOn24 : BOOL ;	//Example for comment: StaOn24WaterPumpA
    StaOn25 : BOOL ;
    StaOn26 : BOOL ;
    StaOn27 : BOOL ;
    StaOn28 : BOOL ;
    StaOn29 : BOOL ;
    StaOn30 : BOOL ;
    StaOn31 : BOOL ;
    StaOn16 : BOOL ;
    StaOn17 : BOOL ;
    StaOn18 : BOOL ;
    StaOn19 : BOOL ;
    StaOn20 : BOOL ;
    StaOn21 : BOOL ;
    StaOn22 : BOOL ;
    StaOn23 : BOOL ;
    StaOn08 : BOOL ;
    StaOn09 : BOOL ;
    StaOn10 : BOOL ;
    StaOn11 : BOOL ;
    StaOn12 : BOOL ;
    StaOn13 : BOOL ;
    StaOn14 : BOOL ;
    StaOn15 : BOOL ;
    StaOn00 : BOOL ;
    StaOn01 : BOOL ;
    StaOn02 : BOOL ;
    StaOn03 : BOOL ;
    StaOn04 : BOOL ;
    StaOn05 : BOOL ;
    StaOn06 : BOOL ;
    StaOn07 : BOOL ;
   END_STRUCT ;
   Switches2 : STRUCT
    StaOn24 : BOOL ;
    StaOn25 : BOOL ;
    StaOn26 : BOOL ;
    StaOn27 : BOOL ;
    StaOn28 : BOOL ;
    StaOn29 : BOOL ;
    StaOn30 : BOOL ;
    StaOn31 : BOOL ;
    StaOn16 : BOOL ;
    StaOn17 : BOOL ;
    StaOn18 : BOOL ;
    StaOn19 : BOOL ;
    StaOn20 : BOOL ;
    StaOn21 : BOOL ;
    StaOn22 : BOOL ;
    StaOn23 : BOOL ;
    StaOn08 : BOOL ;
    StaOn09 : BOOL ;
    StaOn10 : BOOL ;
    StaOn11 : BOOL ;
    StaOn12 : BOOL ;
    StaOn13 : BOOL ;
    StaOn14 : BOOL ;
    StaOn15 : BOOL ;
    StaOn00 : BOOL ;
    StaOn01 : BOOL ;
    StaOn02 : BOOL ;
    StaOn03 : BOOL ;
    StaOn04 : BOOL ;
    StaOn05 : BOOL ;
    StaOn06 : BOOL ;
    StaOn07 : BOOL ;
   END_STRUCT ;
   Values1 : STRUCT 	//Lineparameter data written by Host-System
    Value01 : DINT ;	//Example for comment: TurnoverTime [xxxs]
    Value02 : DINT ;
    Value03 : DINT ;
    Value04 : DINT ;
    Value05 : DINT ;
    Value06 : DINT ;
    Value07 : DINT ;
    Value08 : DINT ;
    Value09 : DINT ;
    Value10 : DINT ;
    Value11 : DINT ;
    Value12 : DINT ;
    Value13 : DINT ;
    Value14 : DINT ;
    Value15 : DINT ;
    Value16 : DINT ;
    Value17 : DINT ;
    Value18 : DINT ;
    Value19 : DINT ;
    Value20 : DINT ;
    Value21 : DINT ;
    Value22 : DINT ;
    Value23 : DINT ;
    Value24 : DINT ;
    Value25 : DINT ;
    Value26 : DINT ;
    Value27 : DINT ;
    Value28 : DINT ;
    Value29 : DINT ;
    Value30 : DINT ;
   END_STRUCT ;
   FlagSec : STRUCT
    Flag00 : BOOL ;
    Flag001 : BOOL ;
    Flag002 : BOOL ;
    Flag003 : BOOL ;
    Flag004 : BOOL ;
    Flag005 : BOOL ;
    Flag006 : BOOL ;
    Flag007 : BOOL ;
    Flag008 : BOOL ;
    Flag009 : BOOL ;
    Flag0010 : BOOL ;
    Flag0011 : BOOL ;
    Flag0012 : BOOL ;
    Flag0013 : BOOL ;
    Flag0014 : BOOL ;
    Flag0015 : BOOL ;
    Flag0016 : BOOL ;
    Flag0017 : BOOL ;
    Flag0018 : BOOL ;
    Flag0019 : BOOL ;
    Flag0020 : BOOL ;
    Flag0021 : BOOL ;
    Flag0022 : BOOL ;
    Flag0023 : BOOL ;
    Flag0024 : BOOL ;
    Flag0025 : BOOL ;
    Flag0026 : BOOL ;
    Flag0027 : BOOL ;
    Flag0028 : BOOL ;
    Flag0029 : BOOL ;
    Flag0030 : BOOL ;
    FaultDB_Copy : BOOL ;	//Fault DB Copy FC49
   END_STRUCT ;
   FlagGen : STRUCT
    WindAlarm : BOOL ;	//Wind speed is too high
    TurningStarted : BOOL ;	//Germination turning is started
    Flag002 : BOOL ;
    WetStep : BOOL ;	//Active Step is Wet Step
    Flag004 : BOOL ;
    Flag005 : BOOL ;
    Flag006 : BOOL ;
    Flag007 : BOOL ;
    LOAD_VAL_HUB1 : BOOL ;	//Counter lifting device 1
    LOAD_VAL_HUB2 : BOOL ;	//Counter lifting device 2
    LOAD_VAL_DRIVE : BOOL ;	//Counter driving device
    LOAD_VAL_AFTER_FAILURE : BOOL ;	//Counter saved datas after failure
    Flag0012 : BOOL ;
    Flag0013 : BOOL ;
    Flag0014 : BOOL ;
    Flag0015 : BOOL ;
    InterlockedFunktionMode : BOOL ;	//Interlocked Funktion Mode (ILO-Mode) is aktive
    ILO_CmdResetFault : BOOL ;
    Flag0018 : BOOL ;
    Flag0019 : BOOL ;
    Flag0020 : BOOL ;
    Flag0021 : BOOL ;
    Flag0022 : BOOL ;
    Flag0023 : BOOL ;
    Flag0024 : BOOL ;
    Flag0025 : BOOL ;
    Flag0026 : BOOL ;
    Flag0027 : BOOL ;
    Flag0028 : BOOL ;
    Flag0029 : BOOL ;
    Flag0030 : BOOL ;
    Flag0031 : BOOL ;
   END_STRUCT ;
   Spare140 : ARRAY  [148 .. 199 ] OF BYTE ;
   ParIntProcess : STRUCT 	//Processparameter data
    UnloadungRounds : INT  := 2;
    LoadungRounds : INT  := 2;	//
    LoadingOverlap : INT  := 100;	//overlap in xx.x° by loading
    UnloadingOverlap : INT  := 200;	//overlap in xx.x° by unloading
    TargetTimeCleaning : INT ;	//Target time cleaning conveyance in min. [particular NPR]
    ActualTimeCleaning : INT ;	//Actual time cleaning conveyance in min. [particular NPR]
    Value7 : INT ;
    Value8 : INT ;
    Value9 : INT ;
    Value10 : INT ;
    Value11 : INT ;
    Value12 : INT ;
    Value13 : INT ;
    ProcessActivVisuKiln : INT ;	//Display that Process is Active
    StateWordKiln : INT ;	//State-Number of the active Step
    SpeedVentilatorBasic : INT ;	//Setpoint Fanspeed in %
    PosExhaustAirFlapBasic : INT ;	//Setpoint basic flap position in %
    PosRecAirExKilnFlapBasic : INT ;	//Setpoint basic flap position in %
    PosRecAirConChFlapBasic : INT ;	//Setpoint basic flap position in %
    PosFreshAirFlapBasic : INT ;	//Setpoint basic flap position in %
    PosRecycAirFlapBasic : INT ;	//Setpoint basic flap position in %
    Value22 : INT ;
    Value23 : INT ;
    Sollwert_Brenner1 : INT ;	//Setpoint Brenner 1 in %
    Sollwert_Brenner2 : INT ;	//Setpoint Brenner 2 in %
    Sollwert_Brenner3 : INT ;	//Setpoint Brenner 3 in %
    Sollwert_Brenner4 : INT ;	//Setpoint Brenner 4 in %
    ActValueTemperature_R1 : INT ;
    ActValueTemperature_R2 : INT ;
    ActValueTemperature_R3 : INT ;
    ActValueTemperature_R4 : INT ;
    OutputTemRegulator1 : INT ;
    OutputTemRegulator2 : INT ;
    OutputTemRegulator3 : INT ;
    OutputTemRegulator4 : INT ;
    Speed_ILO_FloorRotating : INT  := 22;	//Rotating speed floor from ILO-Rotating Floor Drives
    Speed_ILO_UnderCleaning : INT  := 80;	//Rotating speed floor from ILO-Floor Cleaning from below
    Speed_ILO_WallCleaning : INT  := 80;	//Rotating speed floor from ILO-WallCleaning
    TarPos_ILO_1 : INT ;	//Target positon from ILO-Mode
    TarPos_ILO_2 : INT ;	//Target positon from ILO-Mode
    TarPos_ILO_LiftDev : INT ;	//Target positon lifting devices from ILO-Mode
    TarPos_ILO_FreshAir : INT ;	//Target positon fresh air flap from ILO-Mode
    TarPos_ILO_RecycAir : INT ;	//Target positon recycling air flap from ILO-Mode
    Speed_ILO_Fan : INT ;	//Target speed germinatimng fan from ILO-Mode
    Speed_ILO_TravelDrive : INT ;	//Target speed travelling drive from ILO-Mode
    TarPos_ILO_WasteAir : INT ;	//Target positon waste air flap from ILO-Mode
    TargetTemperature_ILO : INT ;	//Target temperature from ILO-Mode
    TarPos_ILO_RecycAirToEx : INT ;	//Target positon recycling air to extern kiln flap from ILO-Mode
    TarPos_ILO_RecycAirToCha : INT ;	//Target positon recycling air to channel between both kiln flap from ILO-Mode
    ActualStep : INT ;	//Actual Step for visu
   END_STRUCT ;
   ParIntMachine : STRUCT 	//Machine parameter data
    ActualStep : INT ;	//Actual process step
    MAX_HUB_DIFF : INT  := 36;	//Max. Hubdifferenz zwischen Hubzug 1 + 2
    REINIGUNGSHOEHE : INT  := 100;	//Reinigungshoehe in mm
    MAX_SCHIEFLAGE : INT  := 150;	//Max. Schieflage zwischen Hubzug 1 + 2
    IMPULSE_HUBZUG1_OBEN : INT  := 480;	//Impulse : Hubantrieb 1 normieren bei Endpos.oben
    IMPULSE_HUBZUG2_OBEN : INT  := 480;	//Impulse : Hubantrieb 2 normieren bei Endpos.oben
    POSITION_HUBZUG1_OBEN : INT  := 1055;	//Hoehe in mm
    POSITION_HUBZUG2_OBEN : INT  := 1055;	//Hoehe in mm
    IMPULSE_RUNDE : INT  := 816;	//Impulse : Fahrantriebantrieb eine Runde (Diesen Wert bei der IBS ermitteln!!)
    SollwertFahrantrWenden : WORD  := W#16#DEF;	//21,7% von 100 Hz
    LiftDevMinPos : INT  := 100;	//Lifting device minimal position for rotation backwards
    FUELLHOEHE_PRODUKT : INT ;	//Produkt-Füllhöhe
    SollpositionFahrantrieb : INT ;	//Soll-Position Fahrantrieb im Prozess
    Value14 : INT ;
    Value15 : INT ;
    LoadingLevelRound_4 : INT ;	//Calculated value level in 4. round
    LoadingLevelRound_5 : INT ;	//Calculated value level in 5. round
    LoadingLevelRound_6 : INT ;	//Calculated value level in 6. round
    LiftingPositionRound_4 : INT ;	//Calculated value lifting position in loading round 4
    LiftingPositionRound_5 : INT ;	//Calculated value lifting position in loading round 5
    LiftingPositionRound_6 : INT ;	//Calculated value lifting position in loading round 6
    Value22 : INT ;
    Value23 : INT ;
    Value24 : INT ;
    Value25 : INT ;
    TargetPosWasteAirLouvers : INT ;
    Value27 : INT ;
    Value28 : INT ;
    Value29 : INT ;
    Value30 : INT ;
    KilningBoxNumber : INT ;
    Value32 : INT ;
    Value33 : INT ;
    Value34 : INT ;
    Value35 : INT ;
    Value36 : INT ;
    Value37 : INT ;
    Value38 : INT ;
    Value39 : INT ;
    Value40 : INT ;
    Value41 : INT ;
    Value42 : INT ;
    Value43 : INT ;
    Value44 : INT ;
    Value45 : INT ;
    Value46 : INT ;
    Value47 : INT ;
    Value48 : INT ;
    Value49 : INT ;
    LastLoadingLevel : INT ;	//saved loading value
   END_STRUCT ;
   FlagFunction_0 : STRUCT 	//Flags section
    Inf24 : BOOL ;	//Example for comment: Inf24WaterPumpA
    LoadingFirstPartEnd : BOOL ;	//End of loading first part from germinating box
    LoadingSecondPartEnd : BOOL ;	//End of loading second part from germinating box
    ReducedSpeed : BOOL ;	//Reduced speed geminating box
    TimeCleanConvRun : BOOL ;	//Time cleaning conveyance running [particular NPR]
    Inf29 : BOOL ;
    Inf30 : BOOL ;
    Inf31 : BOOL ;
    ManualUnloading_Impuls : BOOL ;
    ManualUnloading_Select : BOOL ;
    ManualUnloading_Start : BOOL ;
    AutostartAbraeumenFP : BOOL ;
    AutostartAbraeumen : BOOL ;
    MerkerBeladenGestartet : BOOL ;
    MerkerEntladenGestartet : BOOL ;
    MerkerBeladenGestartetFP : BOOL ;
    ImpulsBeladenGestartet : BOOL ;
    MerkerEntladGestartetFP : BOOL ;
    ImpulsEntladenGestartet : BOOL ;
    MerkerSollpositionFP : BOOL ;
    ImpulsSollposition : BOOL ;
    Inf13 : BOOL ;
    Inf14 : BOOL ;
    Inf15 : BOOL ;
    LoadingLevelNextRound : BOOL ;
    ImpulsUnloadLevelReached : BOOL ;	//ImpulsUnloadLevelReached
    UnloadLevelReachedFP : BOOL ;	//UnloadLevelReachedFP
    OverlapSaved : BOOL ;	//Ueberlappung erfasst
    Inf04 : BOOL ;
    Inf05 : BOOL ;
    ScrewAboveProductLayer : BOOL ;	//Schnecke hat die Produktschichthoehe nicht erreicht
    Inf07 : BOOL ;
   END_STRUCT ;
   FlagMachine : STRUCT 	//flags machine funktion
    CmdTurnFwdAfterLoading : BOOL ;	//Turning direction forward to zero point after finish loading
    CmdTurnRevAfterLoading : BOOL ;	//Turning direction reverse to zero point after finish loading
    CmdTurnFwdAfterTurning : BOOL ;	//Turning direction forward to zero point after finish turning
    CmdTurnRevAfterTurning : BOOL ;	//Turning direction reverse to zero point after finish turning
    CmdTurnFwdAfterUnloading : BOOL ;	//Turning direction forward to zero point after finish unloading
    CmdTurnRevAfterUnloading : BOOL ;	//Turning direction reverse to zero point after finish unloading
    Inf30 : BOOL ;
    Inf31 : BOOL ;
    Inf16 : BOOL ;
    Inf17 : BOOL ;
    Inf18 : BOOL ;
    Inf19 : BOOL ;
    Inf20 : BOOL ;
    Inf21 : BOOL ;
    Inf22 : BOOL ;
    Inf23 : BOOL ;
    Inf08 : BOOL ;
    Inf09 : BOOL ;
    Inf10 : BOOL ;
    Fahrantrieb_Speed_Ctr1 : BOOL ;	//Fahrantrieb Drehueberwachung
    Fahrantrieb_Start_ok : BOOL ;	//Es sind weniger als 2 Fahrantriebe nicht gestartet
    Fahrantrieb_FU_Fault : BOOL ;	//Sammelstörung von allen 12 FU's
    Fahrantriebe_Fwd_Rev : BOOL ;	//Aktuelle Drehrichtung Fahrantriebe (0=Fwd; 1=Rev)
    Fahrantriebe_Vorwaerts : BOOL ;	//Fahrantriebe Ausgang Richtung Vorwärts
    Fahrantriebe_Rueckwaerts : BOOL ;	//Fahrantriebe Ausgang Richtung Rückwärts
    NULL_INDEX_FP : BOOL ;	//Back to zero position after finish cleaning [particular NPR]
    ImpulsNullstellung : BOOL ;	//Back to zero position after finish loading [particular NPR]
    ImpulsNullstellungFP : BOOL ;	//Back to zero position after finish turning [particular NPR]
    WEGMESSUNG_0 : BOOL ;	//Back to zero position after finish unloading [particular NPR]
    WEGMESSUNG_0_FLAG : BOOL ;	//Flatten after finish loading [particular NPR]
    Inf06 : BOOL ;	//Schnecke ueber Produktschicht
    Inf07 : BOOL ;	//Beide Hubzuege in Parkposition
   END_STRUCT ;
   FlagFunction_1 : STRUCT 	//Flags functions
    StepLoading : BOOL ;	//Function Loading is active
    StepUnloading : BOOL ;	//Function Unloading is active
    StepCleaning : BOOL ;	//Function Cleaning is active
    LoadingBreak : BOOL ;	//Function Loading is interrupted
    UnloadingBreak : BOOL ;	//Function Unloading is interrupted
    CleaningBreak : BOOL ;	//Function Cleaning is interrupted
    FinishLoading : BOOL ;	//Function Loading is finished
    FinishUnloading : BOOL ;	//Function Unloading is finished
    FinishCleaning : BOOL ;	//Function Cleaning is finished
    Inf011 : BOOL ;
    Inf012 : BOOL ;
    Inf013 : BOOL ;
    Runde_1 : BOOL ;	//Fahrantrieb 1.Runde
    Runde_2 : BOOL ;	//Fahrantrieb 2.Runde
    Runde_3 : BOOL ;	//Fahrantrieb 3.Runde
    Runde_4 : BOOL ;	//Fahrantrieb 4.Runde
    Runde_5 : BOOL ;	//Fahrantrieb 5.Runde
    Runde_6 : BOOL ;	//Fahrantrieb 6.Runde
    Inf072 : BOOL ;
    Entladerunden_erreicht : BOOL ;	//Fahrantrieb; Entladerunden erreicht
    Reinigungsrunde_erreicht : BOOL ;	//Fahrantrieb; Reinigungsrunde erreicht
    TurningStart : BOOL ;	//Start turning
    TurningStop : BOOL ;	//Stop turning
    TurningLeft : BOOL ;	//Turning direction left
    TurningRight : BOOL ;	//Turning direction right
    LoadFirstPartEnd : BOOL ;	//Grundschicht ist bedeckt, prozess kann starten
    TurningWithSpraying : BOOL ;	//Turning-round in this step with spraying
    TurningWithoutSpraying : BOOL ;	//Turning-round in this step without spraying
    UnloadEnd : BOOL ;	//Kilning box is unloaded
    LoadEnd : BOOL ;	//Kilning box is loaded
    UnloadFirstPart : BOOL ;	//Loading first part from germinating box
    UnloadSecondPart : BOOL ;	//Loading second part from germinating box
   END_STRUCT ;
   FlagProcess : STRUCT 	//Flags process
    ProcessActive : BOOL ;	//Process is active
    Abdarr_Betrieb_Aktiv : BOOL ;
    Schwelk_Betrieb_Aktiv : BOOL ;
    StartProzess_FP : BOOL ;
    Inf04 : BOOL ;
    Inf05 : BOOL ;
    Inf06 : BOOL ;
    Inf07 : BOOL ;
    Inf08 : BOOL ;
    Inf09 : BOOL ;
    DisableFan1 : BOOL ;	//process without fan 1
    DisableFan2 : BOOL ;	//process without fan 2
    Aussenluft_zu_warm : BOOL ;
    StartProzess_SCAN : BOOL ;
    AirMoistenBelowFloor : BOOL ;	//Moisten air
    PressureRegulAboveFloor : BOOL ;	//Regulate air-pressure
    TurningFloor : BOOL ;	//Turning floor 120 degree
    Inf21 : BOOL ;
    Cooling_Activ : BOOL ;	//Cooling
    FP_SendResultToPIC : BOOL ;
    ProcessEnd : BOOL ;
    Vent_ReglerAusg_Plus : BOOL ;
    Vent_ReglerAusg_PlusFP : BOOL ;
    Vent_ReglerAusg_Minus : BOOL ;
    Vent_ReglerAusg_MinusFP : BOOL ;
    Ventilator_Drehzahl_HH : BOOL ;	//Drehzahlbereich HH [85 - 100%]
    Ventilator_Drehzahl_H : BOOL ;	//Drehzahlbereich  H [65 -  84%]
    Ventilator_Drehzahl_L : BOOL ;	//Drehzahlbereich  L [55 -  64%]
    Ventilator_Drehzahl_LL : BOOL ;	//Drehzahlbereich LL [40 -  54%]
    VentilatorDrehzahlMin : BOOL ;
    VentilatorDrehzahlMax : BOOL ;
    ProgrammSchwelkenDarren : BOOL ;
   END_STRUCT ;
   FlagProcess1 : STRUCT 	//Flags process
    GAS_EIN_BRENNER1 : BOOL ;	//Anforderung Gas für Brenner 1
    GAS_EIN_BRENNER2 : BOOL ;	//Anforderung Gas für Brenner 2
    GAS_EIN_BRENNER3 : BOOL ;	//Anforderung Gas für Brenner 3
    GAS_EIN_BRENNER4 : BOOL ;	//Anforderung Gas für Brenner 4
    Brenner1_Regler_Ein : BOOL ;	//Reglerfreigabe vom Brenner 1 ist EIN
    Brenner2_Regler_Ein : BOOL ;	//Reglerfreigabe vom Brenner 2 ist EIN
    Brenner3_Regler_Ein : BOOL ;	//Reglerfreigabe vom Brenner 3 ist EIN
    Brenner4_Regler_Ein : BOOL ;	//Reglerfreigabe vom Brenner 4 ist EIN
    OutRegler_1_Up : BOOL ;
    OutRegler_1_Down : BOOL ;
    OutRegler_2_Up : BOOL ;
    OutRegler_2_Down : BOOL ;
    OutRegler_3_Up : BOOL ;
    OutRegler_3_Down : BOOL ;
    OutRegler_4_Up : BOOL ;
    OutRegler_4_Down : BOOL ;
    HilfsRegler_1_Down : BOOL ;
    HilfsRegler_2_Down : BOOL ;
    HilfsRegler_3_Down : BOOL ;
    HilfsRegler_4_Down : BOOL ;
    Brenner_1_Max : BOOL ;	//Brenner 1: Max. Begrenzung des PID-Schrittreglers
    Brenner_1_Min : BOOL ;	//Brenner 1: Min. Begrenzung des PID-Schrittreglers
    Brenner_2_Max : BOOL ;	//Brenner 2: Max. Begrenzung des PID-Schrittreglers
    Brenner_2_Min : BOOL ;	//Brenner 2: Min. Begrenzung des PID-Schrittreglers
    Brenner_3_Max : BOOL ;	//Brenner 3: Max. Begrenzung des PID-Schrittreglers
    Brenner_3_Min : BOOL ;	//Brenner 3: Min. Begrenzung des PID-Schrittreglers
    Brenner_4_Max : BOOL ;	//Brenner 4: Max. Begrenzung des PID-Schrittreglers
    Brenner_4_Min : BOOL ;	//Brenner 4: Min. Begrenzung des PID-Schrittreglers
    Brenner_1_SPARE : BOOL ;
    Brenner_2_SPARE : BOOL ;
    Brenner_3_SPARE : BOOL ;
    Brenner_4_SPARE : BOOL ;
   END_STRUCT ;
   FlagProcess2 : STRUCT 	//Flags process
    Brenner1_PLUS_Outp_FL : BOOL ;
    Brenner1_PLUS_Outp_FP : BOOL ;
    Brenner1_MINUS_Outp_FL : BOOL ;
    Brenner1_MINUS_Outp_FP : BOOL ;
    Brenner2_PLUS_Outp_FL : BOOL ;
    Brenner2_PLUS_Outp_FP : BOOL ;
    Brenner2_MINUS_Outp_FL : BOOL ;
    Brenner2_MINUS_Outp_FP : BOOL ;
    Brenner3_PLUS_Outp_FL : BOOL ;
    Brenner3_PLUS_Outp_FP : BOOL ;
    Brenner3_MINUS_Outp_FL : BOOL ;
    Brenner3_MINUS_Outp_FP : BOOL ;
    Brenner4_PLUS_Outp_FL : BOOL ;
    Brenner4_PLUS_Outp_FP : BOOL ;
    Brenner4_MINUS_Outp_FL : BOOL ;
    Brenner4_MINUS_Outp_FP : BOOL ;
    Inf20 : BOOL ;
    Inf21 : BOOL ;	//
    Inf22 : BOOL ;	//
    Inf23 : BOOL ;	//
    Inf24 : BOOL ;	//
    Schaltp_15 : BOOL ;	//Temperatur im Brennerraum >15°C
    RegBrennerluftvorw_aktiv : BOOL ;	//Zuheizung Brennerluftvorwärmung
    Schaltp_45 : BOOL ;	//Temperatur unter der Horde >=45°C
    Schaltp_70 : BOOL ;	//Temperatur unter der Horde >=70°C
    Schaltp_5 : BOOL ;	//Temperatur im Brennerraum >5°C
    Freig_Brenner : BOOL ;	//Freigabe Start Brenner
    PosHeizklappe_A : BOOL ;	//Position Heizklappe A <=50%
    PosHeizklappe_B : BOOL ;	//Position Heizklappe B <=50%
    Freig_Brenner_Time : BOOL ;	//Freigabe Brenner nach Zeit T=X
    Freig_Ventilator_A : BOOL ;	//Freigabe Ventilator A wenn Heizklappe A vollstaendig geoeffnet ist
    Freig_Ventilator_B : BOOL ;	//Freigabe Ventilator B wenn Heizklappe B vollstaendig geoeffnet ist
   END_STRUCT ;
   ProcessValue : STRUCT 	//Process values, used only in the PLC
    TemperaturBelowFloor : DINT ;	//Setpoint Temperature in °C
    TemperaturAboveFloor : DINT ;	//Setpoint Temperature in °C
    DeltaTemperatur : DINT ;	//Setpoint Delta-Temperature in °C
    DeltaTemperaturIst : DINT ;	//Delta-Temperature in °C
    MaxTemperaturAboveFloor : DINT ;	//Max. Setpoint Temperature in °C
    Value06 : INT ;
    Value07 : INT ;
    ActMoistureAboveFloor : DINT ;
    ActAirPressureAboveFl : DINT ;
    WasteAirFlapKorr : INT ;
    RecycleAirDoorKorr : INT ;
    RecycleAirJalousKorr : INT ;
    CorrInterval : INT ;	//von Kalle für Brennerregelung verwendet
    Value11 : DINT ;
    Profimess_Command : DINT ;
    Value13 : DINT ;
    Value14 : DINT ;
    Value15 : DINT ;
    Value16 : DINT ;
    Value17 : DINT ;
    Value18 : INT ;
    StepNrActCopy : INT ;
    ActualTimePreviousScan : DATE_AND_TIME ;
    ActualTime : DATE_AND_TIME ;
    BreakPoint : DATE_AND_TIME ;
    StartCooling : DATE_AND_TIME ;
    StepTimeAct : TIME ;
    Afeesttijd : TIME ;
    Value26 : DINT ;
    Value27 : DINT ;
   END_STRUCT ;
   ProcessValue_Real : STRUCT 	//Process real values, used only in the PLC
    SpeedVentilatorBasic : REAL ;	//Setpoint Fanspeed in %
    PositWasteAirFlapBasic : REAL ;	//Setpoint basic flap position
    PositRecyclAirIFlapBasic : REAL ;	//Setpoint basic flap position
    PositRecyclAirDFlapBasic : REAL ;	//Setpoint basic flap position
    Value05 : REAL ;
    Value06 : REAL ;
    Gasmenge_1_R : REAL ;
    Gasmenge_2_R : REAL ;
    Gasmenge_3_R : REAL ;
    Gasmenge_4_R : REAL ;
    GAS1_LITER_PRO_IMPULS : REAL  := 1.000000e+000;	//Gaszähler 1 : Gasmenge [l] pro Impuls
    GAS2_LITER_PRO_IMPULS : REAL  := 1.000000e+000;	//Gaszähler 2 : Gasmenge [l] pro Impuls
    GAS3_LITER_PRO_IMPULS : REAL  := 1.000000e+000;	//Gaszähler 3 : Gasmenge [l] pro Impuls
    GAS4_LITER_PRO_IMPULS : REAL  := 1.000000e+000;	//Gaszähler 4 : Gasmenge [l] pro Impuls
    ReglerBrenner_Gain : REAL ;
    TI_Var_Drehzahl_HiTeil : INT ;
    TI_Var_Drehzahl_LoTeil : INT ;
    SollwertTempKorr : REAL ;
    SollwertTempKorrFaktor : REAL ;
    T_SOLL_NORM : REAL ;	//Normierter Sollwert
    FactorNormalMode : REAL ;	//Normal mode kilning with 2 fans
    FactorEmergModeBurner1 : REAL ;	//Emergency mode kilning with 1 fan burner 1
    FactorEmergModeBurner2 : REAL ;	//Emergency mode kilning with 1 fan burner 2
    FactorEmergModeBurner3 : REAL ;	//Emergency mode kilning with 1 fan burner 3
    FactorEmergModeBurner4 : REAL ;	//Emergency mode kilning with 1 fan burner 4
    Profimess_Wirkleistung : REAL ;
    Profimess_Blindleistung : REAL ;
    Profimess_Frequenz : REAL ;
    Profimess_Wirkleist_Psec : REAL ;
    Profimess_Arbeit_Batch : REAL ;
    EnergieKWs : REAL ;
   END_STRUCT ;
   MachineValue : STRUCT 	//Machine values, used only in the PLC
    ISTWERT_FAHRANTRIEB_POSI : INT ;	//Ist-Position Fahrantrieb
    FAHRANTRIEB_UMDREHUNGEN : INT ;	//Rundenzaehler Fahrantrieb
    IST_HUB_DIFF : INT ;	//Istwert Hubdifferenz zwischen Hubzug 1 + 2
    ISTWERT_HUBZUG1_Z_IMP : INT ;	//Istwert Zaehlimpulse Hubzug 1
    ISTWERT_HUBZUG2_Z_IMP : INT ;	//Istwert Zaehlimpulse Hubzug 2
    SCHRAEGE_HUB1_HUB2 : INT ;	//Schraege Hub 1 > Hub 2
    SOLLWERT_HUBZUG1_HOEHE : INT ;
    SOLLWERT_HUBZUG2_HOEHE : INT ;
    ISTWERT_HUBZUG1_HOEHE : INT ;
    ISTWERT_HUBZUG2_HOEHE : INT ;
    SCHRAEGE_HUB1_MINUS_HUB2 : INT ;	//Schraege Hub 1 minus Hub 2
    SCHRAEGE_HUB2_MINUS_HUB1 : INT ;	//Schraege Hub 2 minus Hub 1
    BELADERUNDEN_START_HUB : INT ;	//Anhebeposition in Grad
    ISTWERT_FAHRANTRIE_Z_IMP : INT ;	//Istwert Zaehlimpulse Fahrantrieb
    Fahrantriebe_Gestartet : INT ;	//Zaehlwert der gestarteten Fahrantriebe
    SollwertFahrantrieb : WORD ;
    Fahrzeit_Reinigungswagen : INT ;	//Fahrzeit des Reinigungswagens unter der Horde
    Position_Reinigungswagen : INT ;	//Position der Reinigungswagens unter der Horde
    ISTWERT_HUBZUG1_DOPPEL : DINT ;	//Hubzug 1 : Hoehe [mm] Rechenwert
    ISTWERT_HUBZUG2_DOPPEL : DINT ;	//Hubzug 2 : Hoehe [mm] Rechenwert
    BELADERUNDEN_HUB_IMP : DINT ;	//Anhebeposition in Pulsen
    FAHR_GRAD_DOPPEL : DINT ;	//Fahrantrieb : Umdrehung in Grad Rechenwert
    RotatingSpeed : DINT ;	//Rotating Speed temp
    FloorPositionPercent : DINT ;	//Floor position percentagewise
    ResultGasConsumpBurner1 : DINT ;
    ResultGasConsumpBurner2 : DINT ;
    ResultGasConsumpBurner3 : DINT ;
    ResultGasConsumpBurner4 : DINT ;
    ResultWaterConsumption : DINT ;
    ResultEnergyConsumption : DINT ;
    CMDEnergyCountingDevice : DINT ;
    Value23 : DINT ;
    Value24 : DINT ;
    Value25 : DINT ;
    Value26 : DINT ;
    Value27 : DINT ;
    HUBZUG1_Z_IMP_HOLD : DINT ;	//Istwert Zaehlimpulse Hubzug 1 gespeichert
    HUBZUG2_Z_IMP_HOLD : DINT ;	//Istwert Zaehlimpulse Hubzug 2 gespeichert
    FAHRANTRIEB_Z_IMP_HOLD : DINT ;	//Istwert Zaehlimpulse Fahrantrieb gespeichert
   END_STRUCT ;
   MachineValueReal : STRUCT 	//Machine real values, used only in the PLC
    HUB1_MM_PRO_IMPULS : REAL  := 2.197917e+000;	//Hubzug 1 : Hoehe [mm] pro Hubimpuls
    HUB2_MM_PRO_IMPULS : REAL  := 2.197917e+000;	//Hubzug 2 : Hoehe [mm] pro Hubimpuls
    FAHRANTRIEB_IMP_GRAD : REAL  := 4.411765e-001;	//Winkelgrad pro Fahrimpuls (wird automatisch berechnet)
    FAHR_GRAD_PRO_IMPULS : REAL ;	//Fahrantrieb : Umdrehung in Grad pro Fahrimpuls Real-Rechenwert
    IMPULSE_RUNDE_REAL : REAL ;	//Impulse : Fahrantriebantrieb eine Runde Real-Rechenwert
    Faktor_Reinigungswagen_R : REAL ;	//Weg/Zeit-Faktor Reinigungswagens unter der Horde
    Fahrzeit_Reinigungswag_R : REAL ;	//Fahrzeit der Reinigungswagens unter der Horde
    Position_Reinigungswag_R : REAL ;	//Position der Reinigungswagens unter der Horde
    FAHRANTRIEB_IMP_PROZ : REAL ;	//Prozentzahl pro Fahrimpuls (wird automatisch berechnet)
    BELADERUNDEN_START_HUB : REAL ;	//Anhebeposition von % in Grad
    Value11 : REAL ;
    Value12 : REAL ;
    Value13 : REAL ;
    Value14 : REAL ;
    Value15 : REAL ;
    Value16 : REAL ;
    Value17 : REAL ;
    Value18 : REAL ;
    Value19 : REAL ;
    Value20 : REAL ;
    Value21 : REAL ;
    Value22 : REAL ;
    SP_INT_BURNER_1 : REAL ;	//Internal setpoint burner 1
    SP_INT_BURNER_2 : REAL ;	//Internal setpoint burner 2
    SP_INT_BURNER_3 : REAL ;	//Internal setpoint burner 3
    SP_INT_BURNER_4 : REAL ;	//Internal setpoint burner 4
    PV_IN_BURNER_1 : REAL ;	//PROCESS VARIABLE IN / burner 1
    PV_IN_BURNER_2 : REAL ;	//PROCESS VARIABLE IN / burner 2
    PV_IN_BURNER_3 : REAL ;	//PROCESS VARIABLE IN / burner 3
    PV_IN_BURNER_4 : REAL ;	//PROCESS VARIABLE IN / burner 4
   END_STRUCT ;
   Spare892 : INT ;
   Spare894 : INT ;
   Error : STRUCT
    Value : INT ;
    Bit : BOOL ;
   END_STRUCT ;
  END_STRUCT ;	
END_TYPE

TYPE "SSA_Kiln_Recipe"	// UDT 2302
VERSION : 0.1
  STRUCT
   RecipeHeader : UDT 2304;
   Step : ARRAY  [1 .. 30 ] OF UDT 2305;
  END_STRUCT ;	
END_TYPE

TYPE "SSA_Kiln_Analog"	// UDT 2303
VERSION : 0.1
  STRUCT
   SpeedVentilatorBasic : INT ;	//Setpoint Fanspeed in %
   PositWasteAirFlapBasic : INT ;	//Setpoint basic flap position
   PositRecyclAirIFlapBasic : INT ;	//Setpoint basic flap position
   PositRecyclAirDFlapBasic : INT ;	//Setpoint basic flap position
   spare08 : INT ;
   spare10 : INT ;
   spare12 : INT ;
   spare14 : INT ;
   spare16 : INT ;
   spare18 : INT ;
   spare20 : INT ;
   spare22 : INT ;
   spare24 : INT ;
   spare26 : INT ;
   spare28 : INT ;
   spare30 : INT ;
   spare32 : INT ;
   spare34 : INT ;
   Change : STRUCT
    SpeedVentilatorBasicGer : BOOL ;	//the analog value has change if there is a bit
    PositFreshAirFlapBasic : BOOL ;	//the analog value has change if there is a bit
    NumberOfAeriationLines : BOOL ;	//the analog value has change if there is a bit
    DelayNextValve : BOOL ;	//the analog value has change if there is a bit
    DelayNextAeriationCycle : BOOL ;	//the analog value has change if there is a bit
    SpeedVentilator1 : BOOL ;	//the analog value has change if there is a bit
    SpeedVentilator2 : BOOL ;	//the analog value has change if there is a bit
    SpeedVentilator3 : BOOL ;	//the analog value has change if there is a bit
    SpeedVentilator4 : BOOL ;	//the analog value has change if there is a bit
    DrainTimeWaterAeriation : BOOL ;	//the analog value has change if there is a bit
    DrainTimeWaterCO2Suck : BOOL ;	//the analog value has change if there is a bit
    StartSpraying : BOOL ;	//the analog value has change if there is a bit
    TimeSpraying : BOOL ;	//the analog value has change if there is a bit
    DelaySpraying : BOOL ;	//the analog value has change if there is a bit
    SpeedVentilatorBasicKiln : BOOL ;	//the analog value has change if there is a bit
    PositWasteAirFlapBasic : BOOL ;	//the analog value has change if there is a bit
    PositRecyclAirIFlapBasic : BOOL ;	//the analog value has change if there is a bit
    PositRecyclAirDFlapBasic : BOOL ;	//the analog value has change if there is a bit
    SpeedRotatingFloorDrives : BOOL ;	//the analog value has change if there is a bit
    spare_20 : BOOL ;
    spare_21 : BOOL ;
    spare_22 : BOOL ;
    spare_23 : BOOL ;
    spare_24 : BOOL ;
    spare_25 : BOOL ;
    spare_26 : BOOL ;
    spare_27 : BOOL ;
    spare_28 : BOOL ;
    spare_29 : BOOL ;
    spare_30 : BOOL ;
    spare_31 : BOOL ;
    spare_32 : BOOL ;
   END_STRUCT ;
  END_STRUCT ;	
END_TYPE

TYPE "SSA_Kiln_Recipe_Header"	// UDT 2304
VERSION : 0.1
  STRUCT
   NumberOfSteps : INT  := 24;	//Number of steps
   WarningTempAboveFloor : DINT ;	//Setpoint Temperature in °C
   Duration_Kiln : DINT ;	//Estimated duration Kiln
   SPARE_DINT000 : DINT ;
   SPARE_DINT0001 : DINT ;
   SPARE_DINT0002 : DINT ;
   SPARE_DINT0003 : DINT ;
   SPARE_DINT004 : DINT ;
   SPARE_INT000 : INT ;
   SPARE_INT001 : INT ;
   SPARE_INT002 : INT ;
   SPARE_INT003 : INT ;
   DeselectVentilator : INT ;	//Deselect Ventilator (GMC)
   Loading : UDT 2011;
   Unloading : UDT 2012;
   Cleaning : UDT 2013;
  END_STRUCT ;	
END_TYPE

TYPE "SSA_Kiln_Step"	// UDT 2305
VERSION : 0.1
  STRUCT
   StepNumber : INT  := 1;
   StepType : INT  := 1;	//Type Loading = 0;Withering/Curing = 1;Cooling = 2;Unloading = 4;
   NextStep : INT  := 2;
   StepTime_Min : INT ;	//Minimal Steptime in min
   StepTime_Max : INT ;	//Maximal Steptime in min
   TemperaturBelowFloor : DINT ;	//Setpoint Temperature in °C
   TemperaturAboveFloor : DINT ;	//Setpoint Temperature in °C
   SPARE_DINT00 : DINT ;	//
   AirPressureAboveFloor : DINT ;	//Setpoint air-pressure above floor in hPa
   MoistureBelowFloor : DINT ;	//Setpoint air-moisture below floor in 1.1 %
   SPARE_DINT000 : DINT ;
   MoistureAboveFloor : DINT ;	//Switchpoint air-moisture above floor in 1.1 %
   DeltaTempSwitchpointStep : DINT ;	//Switchpoint Delta Temperature go to next step in °C
   MaxTempAboveFloorStep : DINT ;	//Switchpoint Temperature above floor go to next step in °C
   MoistureAboveFloorStep : DINT ;	//Switchpoint air-moisture above floor go to next step in 1.1 %
   SPARE_DINT001 : DINT ;
   SPARE_DINT002 : DINT ;
   SPARE_DINT003 : DINT ;
   SpeedVentilatorBasic : INT ;	//Setpoint Fanspeed in %
   SpeedVentilatorMaximal : INT ;	//Setpoint Fanspeed in % (not used)
   PosExhaustAirFlapBasic : INT ;	//Setpoint basic flap position
   PosExhaustAirFlapMax : INT ;	//Setpoint maximal flap position (not used)
   PosRecAirExKilnFlapBasic : INT ;	//Setpoint basic flap position (GMC)
   PosRecAirExKilnFlapMax : INT ;	//Setpoint maximal flap position (not used)
   PosRecAirConChFlapBasic : INT ;	//Setpoint basic flap position (GMC)
   PosRecAirConChFlapMax : INT ;	//Setpoint maximal flap position (not used)
   PosFreshAirFlapBasic : INT ;	//Setpoint basic flap position (GMC)
   PosFreshAirFlapMax : INT ;	//Setpoint maximal flap position (not used)
   SPARE_INT002 : INT ;
   SPARE_INT003 : INT ;
   SPARE_INT004 : INT ;
   SPARE_INT005 : INT ;
   AirMoistenBelowFloor : BYTE ;	//Moisten air y/n (1/0)
   PressureRegulAboveFloor : BYTE ;	//Regulate air-pressure y/n (1/0)
   TurningFloor : BYTE ;	//Turning floor 120 degree in this step y/n (1/0)
   SPARE_BYTE000 : BYTE ;	//
   CoolingDown : BYTE ;	//Must set to 1 if step-type = 2 (Cooling)
   SPARE_BYTE001 : BYTE ;	//
   SPARE_BYTE002 : BYTE ;	//
   SPARE_BYTE003 : BYTE ;	//
   SPARE_BYTE004 : BYTE ;	//
   SPARE_BYTE005 : BYTE ;	//
  END_STRUCT ;	
END_TYPE

TYPE "CMDs_ILO_Funktion"	// UDT 8015
VERSION : 0.1
  STRUCT
   ILOMode : INT ;	//Actual Active ILO Mode
   GrCMDManOn : ARRAY  [1 .. 32 ] OF //Set group into manual mode
   BOOL ;
   GrCMDManOff : ARRAY  [1 .. 32 ] OF //Switch back group from manual mode to auto
   BOOL ;
   GrCMDManStart : ARRAY  [1 .. 32 ] OF //Start group in manual mode
   BOOL ;
   GrCMDManAdditional : STRUCT
    Cmd1 : ARRAY  [1 .. 32 ] OF //Additional signals in manual mode (left right, up down, fwd rev)
    BOOL ;
    Cmd2 : ARRAY  [1 .. 32 ] OF //Additional signals in manual mode (left right, up down, fwd rev)
    BOOL ;
    Cmd3 : ARRAY  [1 .. 32 ] OF //Additional signals in manual mode (left right, up down, fwd rev)
    BOOL ;
    Cmd4 : ARRAY  [1 .. 32 ] OF //Additional signals in manual mode (left right, up down, fwd rev)
    BOOL ;
   END_STRUCT ;
   GrCMDManStop : ARRAY  [1 .. 32 ] OF //Stop group in manual mode
   BOOL ;
   GrCMDManFaultReset : ARRAY  [1 .. 32 ] OF //Reset Fault group in manual mode
   BOOL ;
   GrSTMan : ARRAY  [1 .. 32 ] OF //State of group (copy of InOutAutostartMan)
   BOOL ;
   Code_ILO_Funktion0 : INT ;
   Code_ILO_Funktion1 : INT ;
   Code_ILO_Funktion2 : INT ;
   Code_ILO_Funktion3 : INT ;
   Code_ILO_Funktion4 : INT ;
   SetpointInt01 : ARRAY  [1 .. 32 ] OF INT ;
   SetpointInt02 : ARRAY  [1 .. 32 ] OF INT ;
   SetpointInt03 : ARRAY  [1 .. 32 ] OF INT ;
   SetpointInt04 : ARRAY  [1 .. 32 ] OF INT ;
   SetpointDint01 : ARRAY  [1 .. 32 ] OF DINT ;
   SetpointDint02 : ARRAY  [1 .. 32 ] OF DINT ;
   SetpointDint03 : ARRAY  [1 .. 32 ] OF DINT ;
   Flag : STRUCT
    EdgeILOModeOn : BOOL ;
   END_STRUCT ;
  END_STRUCT ;	
END_TYPE

TYPE "SSA_LOG_Value"	// UDT 10005
VERSION : 0.0
  STRUCT
   Header : STRUCT
    SecType : BYTE ;
    Format : BYTE ;
   END_STRUCT ;
   TimeStamp : DATE_AND_TIME ;
   Para_0005 : DINT ;
   Para_0007 : WORD ;
   Para_0008 : WORD ;
   Para_0009 : WORD ;
   Para_0010 : WORD ;
   Para_0011 : WORD ;
   Para_0012 : WORD ;
   Para_0013 : WORD ;
   Para_0014 : WORD ;
   Para_0015 : DINT ;
   Para_0017 : DINT ;
   Para_0019 : DINT ;
   Para_0021 : DINT ;
   Para_0023 : DINT ;
   Para_0025 : DINT ;
   Para_0027 : DINT ;
   Para_0029 : DINT ;
   Para_0031 : DINT ;
   Para_0033 : DINT ;
   Para_0035 : DINT ;
   Para_0037 : DINT ;
   Para_0039 : DINT ;
   Para_0041 : DINT ;
   Para_0043 : DINT ;
   Para_0045 : DINT ;
   Para_0047 : DINT ;
   Para_0049 : DINT ;
   Para_0051 : DINT ;
   Para_0053 : DINT ;
   Para_0055 : DINT ;
   Para_0057 : DINT ;
   Para_0059 : DINT ;
   Para_0061 : DINT ;
   Para_0063 : DINT ;
   Para_0065 : DINT ;
   Para_0067 : DINT ;
   Para_0069 : DINT ;
   Para_0071 : DINT ;
   Para_0073 : DINT ;
   Para_0075 : DINT ;
   Para_0077 : DINT ;
   Para_0079 : DINT ;
   Para_0081 : DINT ;
   Para_0083 : DINT ;
   Para_0085 : DINT ;
   Para_0087 : DINT ;
   Para_0089 : INT ;
   Para_0090 : INT ;
   Para_0091 : INT ;
   Para_0092 : INT ;
   Para_0093 : INT ;
   Para_0094 : INT ;
   Para_0095 : INT ;
   Para_0096 : INT ;
   Para_0097 : INT ;
   Para_0098 : INT ;
   Para_0099 : INT ;
  END_STRUCT ;	
END_TYPE

